VAR_GLOBAL
	//Better have your inputs and outputs!
	// XRTM1
	Serial_stComIn_XRTM1 AT %I* : EL6inData22B; // XRTM1 In Serial Comm Array
	Serial_stComOut_XRTM1 AT %Q* : EL6outData22B; // XRTM1 Out Serual Comm Array
END_VAR

(* stored: Version 1.1.0.1, ProductVersion 3.1.4022.18
   GVL GVL_SerialIO: Id {e2338c89-1965-407c-b604-590f80e0dc24} *)
